{attribute 'pack_mode' := '1'} 
// ------------------------------------------------------------------------- 
//  SRCI Robot Library                                                
// ------------------------------------------------------------------------- 
//                                                                           
//  Object:      DefaultDynamics                                       
//  Author:      Thorsten Brach                                                
//  Date:        2024-06-01
//
//  Description:                                              
//   
//                                                                           
//  Copyright: 
//    (C) 2024 Thorsten Brach. All rights reserved                                                                         
//                                                                           
//  Disclaimer:                                                                           
//    This project is provided without any guarantee and can be used for   
//    private and commercial purposes. Any commercial use is at the user’s 
//    own risk and responsibility.
//
// -------------------------------------------------------------------------
TYPE DefaultDynamics :
STRUCT
  /// Timestamp
  Timestamp        : DT;
  /// Maximum velocity for the axes.
  /// Range [%]: 
  /// •  <0% : Use default velocity given by the user
  /// •   0% : Use internal minimal velocity
  /// • 100% : Use the entire reference velocity, given by the user
  VelocityRate     : REAL;
  /// Maximum acceleration.
  /// Range [%]:
  /// •  <0% : Use default acceleration given by the user
  /// •   0% : Use internal minimal acceleration
  /// • 100% : Use the entire reference acceleration, given by the user
  AccelerationRate : REAL;
  /// Maximum deceleration.
  /// Range [%] : 
  /// •  <0% : Use default deceleration given by the user
  /// •   0% : Use internal minimal deceleration
  /// • 100% : Use the entire reference deceleration, given by the user
  DecelerationRate : REAL;
  /// Maximum jerk
  /// Range [%] : 
  /// •  <0% : Use default jerk given by the user
  /// •   0% : Use internal minimal jerk
  /// • 100% : Use the entire reference jerk, given by the user (Trapezoidal if possible) 
  JerkRate         : REAL;  
END_STRUCT
END_TYPE

{attribute 'pack_mode' := '1'}
// ------------------------------------------------------------------------- 
//  SRCI Robot Library                                                
// ------------------------------------------------------------------------- 
//                                                                           
//  Object:      ReferenceDynamics                                       
//  Author:      Thorsten Brach                                                
//  Date:        2024-06-01
//
//  Description:                                              
//   
//                                                                           
//  Copyright: 
//    (C) 2024 Thorsten Brach. All rights reserved                                                                         
//                                                                           
//  Disclaimer:                                                                           
//    This project is provided without any guarantee and can be used for   
//    private and commercial purposes. Any commercial use is at the user’s 
//    own risk and responsibility.
//
// ------------------------------------------------------------------------- 
TYPE ReferenceDynamics :
STRUCT
  /// Timestamp
  Timestamp             : DT;
  /// Path velocity [mm/s](tangent) at 100%
  /// • <0: (default) - Do not change values
  /// • ≥0: Change values according to input value
  VelocityReference     : REAL;
  /// Path acceleration [mm/s2] at 100%
  /// • <0: (default) - Do not change values
  /// • ≥0: Change values according to input value
  AccelerationReference : REAL;
  /// Path deceleration [mm/s2] at 100%
  /// • <0: (default) - Do not change values
  /// • ≥0: Change values according to input value
  DecelerationReference : REAL;
  /// Jerk [mm/s3] at 100%
  /// • <0: (default) - Do not change values
  /// • ≥0: Change values according to input value
  JerkRate              : REAL;  
END_STRUCT
END_TYPE

{attribute 'pack_mode' := '1'} 
// ------------------------------------------------------------------------- 
//  SRCI Robot Library                                                
// ------------------------------------------------------------------------- 
//                                                                           
//  Object:      RobotJointCurrent                                       
//  Author:      Thorsten Brach                                                
//  Date:        2024-06-01
//
//  Description:                                              
//   
//                                                                           
//  Copyright: 
//    (C) 2024 Thorsten Brach. All rights reserved                                                                         
//                                                                           
//  Disclaimer:                                                                           
//    This project is provided without any guarantee and can be used for   
//    private and commercial purposes. Any commercial use is at the user’s 
//    own risk and responsibility.
//
// -------------------------------------------------------------------------
TYPE RobotJointCurrent :
STRUCT
  /// Current of first joint of the robot
  J1 : REAL;
  /// Current of second joint of the robot
  J2 : REAL;
  /// Current of third joint of the robot
  J3 : REAL;
  /// Current of fourth joint of the robot
  J4 : REAL;
  /// Current of fifth joint of the robot
  J5 : REAL;
  /// Current of sixth joint of the robot
  J6 : REAL;
  /// Current of first external joint of the robot
  E1 : REAL;
  /// Current of second external axis
  E2: REAL;
  /// Current of third external axis
  E3: REAL;
  /// Current of fourth external axis
  E4: REAL;
  /// Current of fifth external axis
  E5: REAL;
  /// Current of sixth external axis
  E6: REAL;  
END_STRUCT
END_TYPE

{attribute 'pack_mode' := '1'} 
// ------------------------------------------------------------------------- 
//  SRCI Robot Library                                                
// ------------------------------------------------------------------------- 
//                                                                           
//  Object:      RobotJointCurrentExt                                       
//  Author:      Thorsten Brach                                                
//  Date:        2024-06-01
//
//  Description:                                              
//   
//                                                                           
//  Copyright: 
//    (C) 2024 Thorsten Brach. All rights reserved                                                                         
//                                                                           
//  Disclaimer:                                                                           
//    This project is provided without any guarantee and can be used for   
//    private and commercial purposes. Any commercial use is at the user’s 
//    own risk and responsibility.
//
// -------------------------------------------------------------------------
TYPE RobotJointCurrentExt :
STRUCT
  /// Current of first external joint of the robot
  E1 : REAL;
  /// Current of second external axis
  E2: REAL;
  /// Current of third external axis
  E3: REAL;
  /// Current of fourth external axis
  E4: REAL;
  /// Current of fifth external axis
  E5: REAL;
  /// Current of sixth external axis
  E6: REAL;  
END_STRUCT
END_TYPE

{attribute 'pack_mode' := '1'} 
// ------------------------------------------------------------------------- 
//  SRCI Robot Library                                                
// ------------------------------------------------------------------------- 
//                                                                           
//  Object:      RobotJointCurrentShort                                       
//  Author:      Thorsten Brach                                                
//  Date:        2024-06-01
//
//  Description:                                              
//   
//                                                                           
//  Copyright: 
//    (C) 2024 Thorsten Brach. All rights reserved                                                                         
//                                                                           
//  Disclaimer:                                                                           
//    This project is provided without any guarantee and can be used for   
//    private and commercial purposes. Any commercial use is at the user’s 
//    own risk and responsibility.
//
// -------------------------------------------------------------------------
TYPE RobotJointCurrentShort :
STRUCT
  /// Current of first joint of the robot
  J1 : REAL;
  /// Current of second joint of the robot
  J2 : REAL;
  /// Current of third joint of the robot
  J3 : REAL;
  /// Current of fourth joint of the robot
  J4 : REAL;
  /// Current of fifth joint of the robot
  J5 : REAL;
  /// Current of sixth joint of the robot
  J6 : REAL;
END_STRUCT
END_TYPE

{attribute 'pack_mode' := '1'} 
// ------------------------------------------------------------------------- 
//  SRCI Robot Library                                                
// ------------------------------------------------------------------------- 
//                                                                           
//  Object:      RobotJointPosition                                       
//  Author:      Thorsten Brach                                                
//  Date:        2024-06-01
//
//  Description:                                              
//   
//                                                                           
//  Copyright: 
//    (C) 2024 Thorsten Brach. All rights reserved                                                                         
//                                                                           
//  Disclaimer:                                                                           
//    This project is provided without any guarantee and can be used for   
//    private and commercial purposes. Any commercial use is at the user’s 
//    own risk and responsibility.
//
// -------------------------------------------------------------------------
TYPE RobotJointPosition :
STRUCT
  /// Position [°] of first joint of the robot
  J1 : REAL;
  /// Position [°] of second joint of the robot
  J2 : REAL;
  /// Position [°] of third joint of the robot
  J3 : REAL;
  /// Position [°] of fourth joint of the robot
  J4 : REAL;
  /// Position [°] of fifth joint of the robot
  J5 : REAL;
  /// Position [°] of sixth joint of the robot
  J6 : REAL;
  /// Position [°] of first external axis 
  E1 : REAL;  
  /// Position [°] of second external axis
  E2 : REAL;
  /// Position [°] of third external axis
  E3 : REAL;
  /// Position [°] of fourth external axis
  E4 : REAL;
  /// Position [°] of fifth external axis
  E5 : REAL;
  /// Position [°] of sixth external axis
  E6 : REAL;  
END_STRUCT
END_TYPE

{attribute 'pack_mode' := '1'} 
// ------------------------------------------------------------------------- 
//  SRCI Robot Library                                                
// ------------------------------------------------------------------------- 
//                                                                           
//  Object:      RobotJointPositionExt                                       
//  Author:      Thorsten Brach                                                
//  Date:        2024-06-01
//
//  Description:                                              
//   
//                                                                           
//  Copyright: 
//    (C) 2024 Thorsten Brach. All rights reserved                                                                         
//                                                                           
//  Disclaimer:                                                                           
//    This project is provided without any guarantee and can be used for   
//    private and commercial purposes. Any commercial use is at the user’s 
//    own risk and responsibility.
//
// -------------------------------------------------------------------------
TYPE RobotJointPositionExt :
STRUCT
  /// Position of second external axis
  E2: REAL;
  /// Position of third external axis
  E3: REAL;
  /// Position of fourth external axis
  E4: REAL;
  /// Position of fifth external axis
  E5: REAL;
  /// Position of sixth external axis
  E6: REAL;  
END_STRUCT
END_TYPE

{attribute 'pack_mode' := '1'} 
// ------------------------------------------------------------------------- 
//  SRCI Robot Library                                                
// ------------------------------------------------------------------------- 
//                                                                           
//  Object:      RobotJointPositionShort                                       
//  Author:      Thorsten Brach                                                
//  Date:        2024-06-01
//
//  Description:                                              
//   
//                                                                           
//  Copyright: 
//    (C) 2024 Thorsten Brach. All rights reserved                                                                         
//                                                                           
//  Disclaimer:                                                                           
//    This project is provided without any guarantee and can be used for   
//    private and commercial purposes. Any commercial use is at the user’s 
//    own risk and responsibility.
//
// -------------------------------------------------------------------------
TYPE RobotJointPositionShort :
STRUCT
  /// Position of first joint of the robot
  J1 : REAL;
  /// Position of second joint of the robot
  J2 : REAL;
  /// Position of third joint of the robot
  J3 : REAL;
  /// Position of fourth joint of the robot
  J4 : REAL;
  /// Position of fifth joint of the robot
  J5 : REAL;
  /// Position of sixth joint of the robot
  J6 : REAL;
  /// Position of first external axis 
  E1 : REAL;  
END_STRUCT
END_TYPE

{attribute 'pack_mode' := '1'} 
// ------------------------------------------------------------------------- 
//  SRCI Robot Library                                                
// ------------------------------------------------------------------------- 
//                                                                           
//  Object:      AlarmMessage                                       
//  Author:      Thorsten Brach                                                
//  Date:        2024-06-01
//
//  Description:                                              
//   
//                                                                           
//  Copyright: 
//    (C) 2024 Thorsten Brach. All rights reserved                                                                         
//                                                                           
//  Disclaimer:                                                                           
//    This project is provided without any guarantee and can be used for   
//    private and commercial purposes. Any commercial use is at the user’s 
//    own risk and responsibility.
//
// -------------------------------------------------------------------------
TYPE AlarmMessage :
STRUCT
  /// Timestamp
  Timestamp   : DT;
  /// Type of message according to Table 5-46:
  MessageType : MessageType;
  /// Severity of message according to Table 5-47: Debug, Info, Warning, Error, Fatal error
  Severity    : Severity;
  /// Code of messages
  MessageCode : DWORD;
  /// Static text of message
  MessageText : STRING(150);  
END_STRUCT
END_TYPE

{attribute 'pack_mode' := '1'} 
// ------------------------------------------------------------------------- 
//  SRCI Robot Library                                                
// ------------------------------------------------------------------------- 
//                                                                           
//  Object:      ArmConfigParameter                                       
//  Author:      Thorsten Brach                                                
//  Date:        2024-06-01
//
//  Description:                                              
//   
//                                                                           
//  Copyright: 
//    (C) 2024 Thorsten Brach. All rights reserved                                                                         
//                                                                           
//  Disclaimer:                                                                           
//    This project is provided without any guarantee and can be used for   
//    private and commercial purposes. Any commercial use is at the user’s 
//    own risk and responsibility.
//
// -------------------------------------------------------------------------
TYPE ArmConfigParameter :
STRUCT
  /// Configuration of shoulder
  Shoulder : ArmConfigShoulder;
  /// Configuration of elbow
  Elbow    : ArmConfigElbow;
  /// Configuration of wrist
  Wrist    : ArmConfigWrist;
END_STRUCT
END_TYPE

{attribute 'pack_mode' := '1'} 
// ------------------------------------------------------------------------- 
//  SRCI Robot Library                                                
// ------------------------------------------------------------------------- 
//                                                                           
//  Object:      AuxOffset                                       
//  Author:      Thorsten Brach                                                
//  Date:        2024-06-01
//
//  Description:                                              
//   
//                                                                           
//  Copyright: 
//    (C) 2024 Thorsten Brach. All rights reserved                                                                         
//                                                                           
//  Disclaimer:                                                                           
//    This project is provided without any guarantee and can be used for   
//    private and commercial purposes. Any commercial use is at the user’s 
//    own risk and responsibility.
//
// -------------------------------------------------------------------------
TYPE AuxOffset :
STRUCT
  /// Offset in X-Direction
  X : REAL;
  /// Offset in Y-direction
  Y : REAL;
  /// Offset in Z-direction
  Z : REAL;
END_STRUCT
END_TYPE

{attribute 'pack_mode' := '1'} 
// ------------------------------------------------------------------------- 
//  SRCI Robot Library                                                
// ------------------------------------------------------------------------- 
//                                                                           
//  Object:      CoordinateSystem                                       
//  Author:      Thorsten Brach                                                
//  Date:        2024-06-01
//
//  Description:                                              
//   
//                                                                           
//  Copyright: 
//    (C) 2024 Thorsten Brach. All rights reserved                                                                         
//                                                                           
//  Disclaimer:                                                                           
//    This project is provided without any guarantee and can be used for   
//    private and commercial purposes. Any commercial use is at the user’s 
//    own risk and responsibility.
//
// -------------------------------------------------------------------------
TYPE CoordinateSystem :
STRUCT
  /// Tool index
  /// • 0: Flange
  /// • 1..254: Tool frames
  ToolNo  : USINT;
  /// Frame index
  /// • 0: WCS
  /// • 1..254: User frames
  FrameNo : USINT;
END_STRUCT
END_TYPE

{attribute 'pack_mode' := '1'} 
// ------------------------------------------------------------------------- 
//  SRCI Robot Library                                                
// ------------------------------------------------------------------------- 
//                                                                           
//  Object:      DataInSync                                       
//  Author:      Thorsten Brach                                                
//  Date:        2024-06-01
//
//  Description:                                              
//   
//                                                                           
//  Copyright: 
//    (C) 2024 Thorsten Brach. All rights reserved                                                                         
//                                                                           
//  Disclaimer:                                                                           
//    This project is provided without any guarantee and can be used for   
//    private and commercial purposes. Any commercial use is at the user’s 
//    own risk and responsibility.
//
// -------------------------------------------------------------------------
TYPE DataInSync :
STRUCT
  /// TRUE, if no tool has been modified
  ToolsInSync             : BOOL;
  /// TRUE, if no frame has been modified
  FramesInSync            : BOOL;
  /// TRUE, if no load has been modified
  LoadsInSync             : BOOL;
  /// TRUE, if no work area has been modified
  WorkAreasInSync         : BOOL;
  /// TRUE, if no software limit has been modified
  SoftwareLimitsInSync    : BOOL;
  /// TRUE, if no default dynamic parameter has been modified
  DefaultDynamicsInSync   : BOOL;
  /// TRUE, if no reference dynamic parameter has been modified
  ReferenceDynamicsInSync : BOOL;  
END_STRUCT
END_TYPE

{attribute 'pack_mode' := '1'} 
// ------------------------------------------------------------------------- 
//  SRCI Robot Library                                                
// ------------------------------------------------------------------------- 
//                                                                           
//  Object:      DHParameter                                       
//  Author:      Thorsten Brach                                                
//  Date:        2024-06-01
//
//  Description:                                              
//   
//                                                                           
//  Copyright: 
//    (C) 2024 Thorsten Brach. All rights reserved                                                                         
//                                                                           
//  Disclaimer:                                                                           
//    This project is provided without any guarantee and can be used for   
//    private and commercial purposes. Any commercial use is at the user’s 
//    own risk and responsibility.
//
// -------------------------------------------------------------------------
TYPE DHParameter :
STRUCT
   /// DH parameter α for each joint - 0 If not supported
   Alpha                  : ARRAY [0..6] OF REAL;
   /// DH parameters A for each joint - 0 If not supported
   A                      : ARRAY [0..6] OF REAL;
   /// DH parameters D for each joint - 0 If not supported
   D                      : ARRAY [0..6] OF REAL;
   /// DH parameters Theta for each joint - 0 If not supported
   Theta                  : ARRAY [0..6] OF REAL;
   /// Positive joint direction of each joint. TRUE when positive joint direction points to the right.
   /// See also Figure 6-16.
   PositiveJointDirection : ARRAY [0..6] OF BOOL;
   /// Offset of zero position of joint to zero position suggested by Figure 6-17.
   JointZeroPosition      : ARRAY [0..6] OF REAL;
END_STRUCT
END_TYPE

{attribute 'pack_mode' := '1'} 
// ------------------------------------------------------------------------- 
//  SRCI Robot Library                                                
// ------------------------------------------------------------------------- 
//                                                                           
//  Object:      ExternalAxesFlags                                       
//  Author:      Thorsten Brach                                                
//  Date:        2024-06-01
//
//  Description:                                              
//   
//                                                                           
//  Copyright: 
//    (C) 2024 Thorsten Brach. All rights reserved                                                                         
//                                                                           
//  Disclaimer:                                                                           
//    This project is provided without any guarantee and can be used for   
//    private and commercial purposes. Any commercial use is at the user’s 
//    own risk and responsibility.
//
// -------------------------------------------------------------------------
TYPE ExternalAxesFlags :
STRUCT
  /// Bit 00 : Not used
  Bit00   : BOOL;
  /// Bit 01 : External axis E1 - property depends of usage 
  AxisE1  : BOOL;
  /// Bit 02 : External axis E2 - property depends of usage 
  AxisE2  : BOOL;
  /// Bit 03 : External axis E3 - property depends of usage 
  AxisE3  : BOOL;
  /// Bit 04 : External axis E4 - property depends of usage 
  AxisE4  : BOOL;
  /// Bit 05 : External axis E5 - property depends of usage 
  AxisE5  : BOOL;
  /// Bit 06 : External axis E6 - property depends of usage 
  AxisE6  : BOOL;
  /// Bit 00 : Not used
  Bit07   : BOOL;
END_STRUCT
END_TYPE

{attribute 'pack_mode' := '1'} 
// ------------------------------------------------------------------------- 
//  SRCI Robot Library                                                
// ------------------------------------------------------------------------- 
//                                                                           
//  Object:      ForceStatus                                       
//  Author:      Thorsten Brach                                                
//  Date:        2024-06-01
//
//  Description:                                              
//   
//                                                                           
//  Copyright: 
//    (C) 2024 Thorsten Brach. All rights reserved                                                                         
//                                                                           
//  Disclaimer:                                                                           
//    This project is provided without any guarantee and can be used for   
//    private and commercial purposes. Any commercial use is at the user’s 
//    own risk and responsibility.
//
// -------------------------------------------------------------------------
TYPE ForceStatus :
STRUCT
  /// TRUE, while a "ForceControl" function is enabled
  ForceControlEnabled         : BOOL;
  /// TRUE, while a "ForceLimit" function is enabled
  ForceLimitEnabled           : BOOL;
  /// TRUE, while robot is adjusting its movement to apply specified force
  ApplyingForce               : BOOL;
  /// TRUE, while maximum deviation according to input parameter "MaxDeviation" is reached
  MaxDeviationReached         : BOOL;
  /// TRUE, while currently applied force/torque is identical to specified force/torque
  SpecifiedForceTorqueReached : BOOL;
  /// TRUE, while currently detected force is identical to specified force limit
  SpecifiedForceLimitReached  : BOOL;
  /// Bit 06 Reserve
  Bit06                       : BOOL;
  /// Bit 07 Reserve
  Bit07                       : BOOL;  
END_STRUCT
END_TYPE

{attribute 'pack_mode' := '1'} 
// ------------------------------------------------------------------------- 
//  SRCI Robot Library                                                
// ------------------------------------------------------------------------- 
//                                                                           
//  Object:      FragmentAction                                       
//  Author:      Thorsten Brach                                                
//  Date:        2024-06-01
//
//  Description:                                              
//   
//                                                                           
//  Copyright: 
//    (C) 2024 Thorsten Brach. All rights reserved                                                                         
//                                                                           
//  Disclaimer:                                                                           
//    This project is provided without any guarantee and can be used for   
//    private and commercial purposes. Any commercial use is at the user’s 
//    own risk and responsibility.
//
// -------------------------------------------------------------------------
TYPE FragmentAction :
STRUCT
  /// Bit 00 : Command Message is completely received – Flag to trigger processing of the payload
  Complete : BOOL;
  /// Bit 01 :(only client->server): The first message fragment of a new CMD resets (set all ACR values of this CMD ID to 0) the ACR entry
  Reset    : BOOL;
  /// Bit 02: Clears the receiving buffer by setting all of its Bytes to 0.
  Clear    : BOOL;
  /// Bit 03
  BIT03    : BOOL;
  /// Bit 04
  BIT04    : BOOL;
  /// Bit 05
  BIT05    : BOOL;
  /// Bit 06
  BIT06    : BOOL;
  /// Bit 07
  BIT07    : BOOL;  
END_STRUCT
END_TYPE

{attribute 'pack_mode' := '1'} 
// ------------------------------------------------------------------------- 
//  SRCI Robot Library                                                
// ------------------------------------------------------------------------- 
//                                                                           
//  Object:      JogControl                                       
//  Author:      Thorsten Brach                                                
//  Date:        2024-06-01
//
//  Description:                                              
//   
//                                                                           
//  Copyright: 
//    (C) 2024 Thorsten Brach. All rights reserved                                                                         
//                                                                           
//  Disclaimer:                                                                           
//    This project is provided without any guarantee and can be used for   
//    private and commercial purposes. Any commercial use is at the user’s 
//    own risk and responsibility.
//
// -------------------------------------------------------------------------
TYPE JogControl :
STRUCT
  /// Mode Frame : Movement in positive direction X of selected frame
  /// Mode Tool  : Movement in positive direction X of selected tool
  /// Mode Axes  : Movement in positive direction joint 1
  X_J1_Pos  : BOOL;
  /// Mode Frame : Movement in negative direction X of selected frame
  /// Mode Tool  : Movement in negative direction X of selected tool
  /// Mode Axes  : Movement in negative direction joint 1
  X_J1_Neg  : BOOL;
  /// Mode Frame : Movement in positive direction Y of selected frame
  /// Mode Tool  : Movement in positive direction Y of selected tool
  /// Mode Axes  : Movement in positive direction joint 2
  Y_J2_Pos  : BOOL;
  /// Mode Frame : Movement in negative direction Y of selected frame
  /// Mode Tool  : Movement in negative direction Y of selected tool
  /// Mode Axes  : Movement in negative direction joint 2
  Y_J2_Neg  : BOOL;
  /// Mode Frame : Movement in positive direction Z of selected frame
  /// Mode Tool  : Movement in positive direction Z of selected tool
  /// Mode Axes  : Movement in positive direction joint 3
  Z_J3_Pos  : BOOL;
  /// Mode Frame : Movement in negative direction Z of selected frame
  /// Mode Tool  : Movement in negative direction Z of selected tool
  /// Mode Axes  : Movement in negative direction joint 3
  Z_J3_Neg  : BOOL;
  /// Mode Frame : Movement in positive direction Rx of selected frame
  /// Mode Tool  : Movement in positive direction Rx of selected tool
  /// Mode Axes  : Movement in positive direction joint 4
  Rx_J4_Pos : BOOL;
  /// Mode Frame : Movement in negative direction Rx of selected frame
  /// Mode Tool  : Movement in negative direction Rx of selected tool
  /// Mode Axes  : Movement in negative direction joint 4
  Rx_J4_Neg : BOOL;
  /// Mode Frame : Movement in positive direction Ry of selected frame
  /// Mode Tool  : Movement in positive direction Ry of selected tool
  /// Mode Axes  : Movement in positive direction joint 5
  Ry_J5_Pos : BOOL;
  /// Mode Frame : Movement in negative direction Ry of selected frame
  /// Mode Tool  : Movement in negative direction Ry of selected tool
  /// Mode Axes  : Movement in negative direction joint 5
  Rx_J5_Neg : BOOL;
  /// Mode Frame : Movement in positive direction Rz of selected frame
  /// Mode Tool  : Movement in positive direction Rz of selected tool
  /// Mode Axes  : Movement in positive direction joint 6
  Rz_J6_Pos : BOOL;
  /// Mode Frame : Movement in negative direction Rz of selected frame
  /// Mode Tool  : Movement in negative direction Rz of selected tool
  /// Mode Axes  : Movement in negative direction joint 6
  Rz_J6_Neg : BOOL;
  /// Mode Frame : not supported
  /// Mode Tool  : not supported
  /// Mode Axes  : Movement in positive direction first external axis
  E1_Pos    : BOOL;
  /// Mode Frame : not supported
  /// Mode Tool  : not supported
  /// Mode Axes  : Movement in negative direction first external axis
  E1_Neg    : BOOL;
  /// Mode Frame : not supported
  /// Mode Tool  : not supported
  /// Mode Axes  : Movement in positive direction second external axis
  E2_Pos    : BOOL;
  /// Mode Frame : not supported
  /// Mode Tool  : not supported
  /// Mode Axes  : Movement in negative direction second external axis
  E2_Neg    : BOOL;
  /// Mode Frame : not supported
  /// Mode Tool  : not supported
  /// Mode Axes  : Movement in positive direction third external axis
  E3_Pos    : BOOL;
  /// Mode Frame : not supported
  /// Mode Tool  : not supported
  /// Mode Axes  : Movement in negative direction third external axis
  E3_Neg    : BOOL;
  /// Mode Frame : not supported
  /// Mode Tool  : not supported
  /// Mode Axes  : Movement in positive direction fourth external axis
  E4_Pos    : BOOL;
  /// Mode Frame : not supported
  /// Mode Tool  : not supported
  /// Mode Axes  : Movement in negative direction fourth external axis
  E4_Neg    : BOOL;
  /// Mode Frame : not supported
  /// Mode Tool  : not supported
  /// Mode Axes  : Movement in positive direction fifth external axis
  E5_Pos    : BOOL;
  /// Mode Frame : not supported
  /// Mode Tool  : not supported
  /// Mode Axes  : Movement in negative direction fifth external axis
  E5_Neg    : BOOL;
  /// Mode Frame : not supported
  /// Mode Tool  : not supported
  /// Mode Axes  : Movement in positive direction sixth external axis
  E6_Pos    : BOOL;
  /// Mode Frame : not supported
  /// Mode Tool  : not supported
  /// Mode Axes  : Movement in negative direction sixts external axis
  E6_Neg    : BOOL;
  
END_STRUCT
END_TYPE

{attribute 'pack_mode' := '1'} 
// ------------------------------------------------------------------------- 
//  SRCI Robot Library                                                
// ------------------------------------------------------------------------- 
//                                                                           
//  Object:      MeasuringInputResult                                       
//  Author:      Thorsten Brach                                                
//  Date:        2024-06-01
//
//  Description:                                              
//   
//                                                                           
//  Copyright: 
//    (C) 2024 Thorsten Brach. All rights reserved                                                                         
//                                                                           
//  Disclaimer:                                                                           
//    This project is provided without any guarantee and can be used for   
//    private and commercial purposes. Any commercial use is at the user’s 
//    own risk and responsibility.
//
// -------------------------------------------------------------------------
TYPE MeasuringInputResult :
STRUCT
  /// Measured robot position value at the rising edge of the digital input in selected coordinate systems (see input parameters ToolNo and FrameNo).
  MeasuredCartesianPosition :  RobotCartesianPosition;
  /// Index of tool of returned position
  /// • 0: Flange
  /// • 1..254: Tool frames
  ToolNo                    : USINT;
  /// Index of frame of returned position
  /// • 0: WCS
  /// • 1..254: User frames
  FrameNo                   : USINT;
  /// Measured robot position value at the rising edge of the digital input in Joint position.
  MeasuredJointPosition     : RobotJointPosition;
END_STRUCT
END_TYPE

{attribute 'pack_mode' := '1'} 
// ------------------------------------------------------------------------- 
//  SRCI Robot Library                                                
// ------------------------------------------------------------------------- 
//                                                                           
//  Object:      ProcessingModeAllowed                                       
//  Author:      Thorsten Brach                                                
//  Date:        2024-06-01
//
//  Description:                                              
//   
//                                                                           
//  Copyright: 
//    (C) 2024 Thorsten Brach. All rights reserved                                                                         
//                                                                           
//  Disclaimer:                                                                           
//    This project is provided without any guarantee and can be used for   
//    private and commercial purposes. Any commercial use is at the user’s 
//    own risk and responsibility.
//
// -------------------------------------------------------------------------
TYPE ProcessingModeAllowed :
STRUCT
  /// Command is buffered in sequence buffer and executed once
  BUFFERED           : BOOL;
  /// Command is buffered in sequence buffer, aborts and empties previous commands in sequence buffer, and is executed once
  ABORTING           : BOOL;
  /// Command is buffered in parallel buffer and executed once
  PARALLEL           : BOOL;
  /// Command is buffered in parallel buffer and executed repeatedly until deliberate deactivation by user
  CONTINUOUS         : BOOL;
  /// CMD execution is stopped and/or CMD is removed from the buffer
  DEACTIVATE         : BOOL;
  /// Command is buffered in sequence buffer and executed once (Trigger based)
  TRIGGER_BUFFERED   : BOOL;
  /// Command is buffered in sequence buffer, aborts and empties previous commands in sequence buffer, and is executed once (Trigger based)
  TRIGGER_ABORTING   : BOOL;
  /// Command is buffered in parallel buffer and executed once (Trigger based)
  TRIGGER_ONCE       : BOOL;
  /// Command is buffered in parallel buffer and executed repeatedly until deliberate deactivation by user (Trigger based)
  TRIGGER_CONTINUOUS : BOOL;
  /// Command is buffered and executed multiple times when triggered. The CMD remains in the buffer until removed by the user.
  TRIGGER_MULTIPLE   : BOOL;  
END_STRUCT
END_TYPE

{attribute 'pack_mode' := '1'} 
// ------------------------------------------------------------------------- 
//  SRCI Robot Library                                                
// ------------------------------------------------------------------------- 
//                                                                           
//  Object:      RaStatusWord                                       
//  Author:      Thorsten Brach                                                
//  Date:        2024-06-01
//
//  Description:                                              
//   
//                                                                           
//  Copyright: 
//    (C) 2024 Thorsten Brach. All rights reserved                                                                         
//                                                                           
//  Disclaimer:                                                                           
//    This project is provided without any guarantee and can be used for   
//    private and commercial purposes. Any commercial use is at the user’s 
//    own risk and responsibility.
//
// -------------------------------------------------------------------------
TYPE RaStatusWord :
STRUCT
  /// Bit 00: 
  /// TRUE, when robot’s axes values change due to physical movement of axes
  IsMoving                 : BOOL;
  /// Bit 01: 
  /// TRUE, when move commands buffered by the primary sequence are currently not processed
  PrimarySequencePaused    : BOOL;
  /// Bit 02: 
  /// TRUE, when robot is moving in the primary sequence, FALSE when robot leaves its position by other means
  /// Switches back to TRUE in the following two scenarios:
  /// 1. During a change to the primary sequence the current TCP position is equal to
  ///    - position when the primary sequence was left
  ///    - target position of an interrupted move command of the primary sequence (see "ReturnToPrimary": "ReturnMode" "End position" chapter 6.3.11)
  /// 2. The primary sequence is active, and the buffer is empty while a new command is buffered by the primary sequence
  /// Independent of RA state
  InPrimaryPos             : BOOL;
  /// Bit 03:
  /// Secondary sequence is active, either by user selection or by implicit behavior
  SecondarySequenceActive  : BOOL;
  /// Bit 04:
  /// TRUE, when robot is currently blending between two move commands
  IsBlending               : BOOL;
  /// Bit 05:
  /// Shows that an error acknowledgement by the client is necessary
  ErrorPending             : BOOL;
  /// Bit 06:
  /// RC is restarting
  RestartInProgress        : BOOL;
  /// Bit 07:
  /// RA power state
  Enabled                  : BOOL;
  /// Bit 08:
  /// RA sequence states: Idle, Interrupt active, Axes controlled
  Executing                : BOOL;
  /// Bit 09:
  /// Interrupted
  Interrupted              : BOOL;
  /// Bit 10 - Bit 12:
  /// Operation Mode: T1 Local, T2 Local, Auto, Auto Ext, T1 Ext, T2 Ext
  OperationMode            : OperationMode;
  /// Bit 13:
  /// TRUE, while CollisionDetection is enabled (see chapter 6.5.35) 
  CollisionDetectedEnabled : BOOL;
  /// Bit 14:
  /// TRUE, when a collision was detected while CollisionDetection is enabled
  CollisionDetected        : BOOL;
  /// Bit 15:
  /// TRUE, when the RC request a restart of the RCinduced through the functions "WriteRobotSWLimits" or "WriteSystemVariable"
  RestartRequested         : BOOL;
  /// Bit 16:
  /// RA is currently accelerating. Support of this value is returned via exchangeConfig.
  Accelerating             : BOOL;
  /// Bit 17:
  /// RA is currently decelerating. Support of this value is returned via exchangeConfig.
  Decelerating             : BOOL;
  /// Bit 18:
  /// RA is currently not accelerating nor decelerating. Support of this value is returned via exchangeConfig.
  ConstantVelocity         : BOOL;
  /// Bit 19
  Bit19                    : BOOL;
  /// Bit 20
  Bit20                    : BOOL;
  /// Bit 21
  Bit21                    : BOOL;
  /// Bit 22
  Bit22                    : BOOL;
  /// Bit 23
  Bit23                    : BOOL;
  /// Bit 24
  Bit24                    : BOOL;
  /// Bit 25
  Bit25                    : BOOL;
  /// Bit 26
  Bit26                    : BOOL;
  /// Bit 27
  Bit27                    : BOOL;
  /// Bit 28
  Bit28                    : BOOL;
  /// Bit 29
  Bit29                    : BOOL;
  /// Bit 30
  Bit30                    : BOOL;
  /// Bit 31
  Bit31                    : BOOL;  
END_STRUCT
END_TYPE

{attribute 'pack_mode' := '1'} 
// ------------------------------------------------------------------------- 
//  SRCI Robot Library                                                
// ------------------------------------------------------------------------- 
//                                                                           
//  Object:      RCSupportedFunctions                                       
//  Author:      Thorsten Brach                                                
//  Date:        2024-06-01
//
//  Description:                                              
//   
//                                                                           
//  Copyright: 
//    (C) 2024 Thorsten Brach. All rights reserved                                                                         
//                                                                           
//  Disclaimer:                                                                           
//    This project is provided without any guarantee and can be used for   
//    private and commercial purposes. Any commercial use is at the user’s 
//    own risk and responsibility.
//
// -------------------------------------------------------------------------
TYPE RCSupportedFunctions :
STRUCT
  /// Byte 00 - Bit 0  
  Reserved                   : BOOL;
  /// Byte 00 - Bit 1 
  ReadRobotData              : BOOL;
  /// Byte 00 - Bit 2  
  EnableRobot                : BOOL;
  /// Byte 00 - Bit 3  
  GroupReset                 : BOOL;
  /// Byte 00 - Bit 4  
  ReadActualPosition         : BOOL;
  /// Byte 00 - Bit 5 
  ReadActualPositionCyclic   : BOOL;
  /// Byte 00 - Bit 6  
  ExchangeConfiguration      : BOOL;
  /// Byte 00 - Bit 7  
  SetSequence                : BOOL;
  
  /// Byte 01 - Bit 0  
  ChangeSpeedOverride        : BOOL;
  /// Byte 01 - Bit 1  
  ReadMessages               : BOOL;
  /// Byte 01 - Bit 2  
  ReadRobotReferenceDynamics : BOOL;
  /// Byte 01 - Bit 3  
  WriteFrameData             : BOOL;
  /// Byte 01 - Bit 4  
  WriteToolData              : BOOL;
  /// Byte 01 - Bit 5  
  WriteLoadData              : BOOL;
  /// Byte 01 - Bit 6  
  WriteRobotReferenceDynamics: BOOL;
  /// Byte 01 - Bit 7  
  WriteRobotDefaultDynamics  : BOOL;
  
  /// Byte 02 - Bit 0  
  ReadRobotDefaultDynamics   : BOOL;
  /// Byte 02 - Bit 1  
  ReadFrameData              : BOOL;
  /// Byte 02 - Bit 2  
  ReadToolData               : BOOL;
  /// Byte 02 - Bit 3  
  ReadLoadData               : BOOL;
  /// Byte 02 - Bit 4  
  ReadRobotSWLimits          : BOOL;
  /// Byte 02 - Bit 5  
  GroupJog                   : BOOL;
  /// Byte 02 - Bit 6  
  MoveLinearAbsolute         : BOOL;
  /// Byte 02 - Bit 7  
  MoveDirectAbsolute         : BOOL;
  
  /// Byte 03 - Bit 0  
  MoveAxesAbsolute           : BOOL;
  /// Byte 03 - Bit 1  
  GroupStop                  : BOOL;
  /// Byte 03 - Bit 2
  GroupContinue              : BOOL;
  /// Byte 03 - Bit 3
  GroupInterrupt             : BOOL;
  /// Byte 03 - Bit 4
  ReturnToPrimary            : BOOL;
  /// Byte 03 - Bit 5
  MoveLinearAbsoluteJ        : BOOL;
  /// Byte 03 - Bit 6
  MoveDirectRelative         : BOOL;
  /// Byte 03 - Bit 7
  MoveAxesRelative           : BOOL;
  
  /// Byte 04 - Bit 0
  MoveCircularAbsolute       : BOOL;
  /// Byte 04 - Bit 1
  MoveCircularRelative       : BOOL;
  /// Byte 04 - Bit 2
  MoveLinearOffset           : BOOL;
  /// Byte 04 - Bit 3
  MoveDirectOffset           : BOOL;
  /// Byte 04 - Bit 4
  WaitTime                   : BOOL;
  /// Byte 04 - Bit 5
  ReadDigitalInputs          : BOOL;
  /// Byte 04 - Bit 6
  ReadDigitalOutputs         : BOOL;
  /// Byte 04 - Bit 7
  WriteDigitalOutputs        : BOOL;
  
  /// Byte 05 - Bit 0
  ReadIntegers               : BOOL;
  /// Byte 05 - Bit 1
  ReadReals                  : BOOL;
  /// Byte 05 - Bit 2
  WriteIntegers              : BOOL;
  /// Byte 05 - Bit 3
  WriteReals                 : BOOL;
  /// Byte 05 - Bit 4
  MoveLinearCam              : BOOL;
  /// Byte 05 - Bit 5
  MoveDirectCam              : BOOL;
  /// Byte 05 - Bit 6
  MoveCircularCam            : BOOL;
  /// Byte 05 - Bit 7
  SetTriggerRegister         : BOOL;
  
  /// Byte 06 - Bit 0
  SetTriggerLimit            : BOOL;
  /// Byte 06 - Bit 1
  SetTriggerUser             : BOOL;
  /// Byte 06 - Bit 2
  SetTriggerError            : BOOL;
  /// Byte 06 - Bit 3
  ReactAtTrigger             : BOOL;
  /// Byte 06 - Bit 4
  WaitForTrigger             : BOOL;
  /// Byte 06 - Bit 5
  ReadSystemVariable         : BOOL;
  /// Byte 06 - Bit 6
  WriteSystemVariable        : BOOL;
  /// Byte 06 - Bit 7
  CalculateForwardKinematic  : BOOL;
  
  /// Byte 07 - Bit 0
  CalculateInverseKinematic  : BOOL;
  /// Byte 07 - Bit 1
  CalculateCartesianPosition : BOOL;
  /// Byte 07 - Bit 2
  CalculateTool              : BOOL;
  /// Byte 07 - Bit 3
  CalculateFrame             : BOOL;
  /// Byte 07 - Bit 4
  ActivateNextCommand        : BOOL;
  /// Byte 07 - Bit 5
  ShiftPosition              : BOOL;
  /// Byte 07 - Bit 6
  CallSubprogram             : BOOL;
  /// Byte 07 - Bit 7
  MoveLinearRelative         : BOOL;
  
  /// Byte 08 - Bit 0
  WriteCallSubprogramCyclic  : BOOL;
  /// Byte 08 - Bit 1
  ReadCallSubprogramCyclic   : BOOL;
  /// Byte 08 - Bit 2
  StopSubprogram             : BOOL;
  /// Byte 08 - Bit 3
  ReadDHParameter            : BOOL;
  /// Byte 08 - Bit 4
  RestartController          : BOOL;
  /// Byte 08 - Bit 5
  ReadActualTCPVelocity      : BOOL;
  /// Byte 08 - Bit 6
  UserLogin                  : BOOL;
  /// Byte 08 - Bit 7
  SwitchLanguage             : BOOL;
  
  /// Byte 09 - Bit 0
  WriteRobotSWLimits         : BOOL;
  /// Byte 09 - Bit 1
  SetOperationMode           : BOOL;
  /// Byte 09 - Bit 2
  ReadWorkArea               : BOOL;
  /// Byte 09 - Bit 3
  WriteWorkArea              : BOOL;
  /// Byte 09 - Bit 4
  ActivateWorkArea           : BOOL;
  /// Byte 09 - Bit 5
  MonitorWorkArea            : BOOL;
  /// Byte 09 - Bit 6
  MoveApproachLinear         : BOOL;
  /// Byte 09 - Bit 7
  MoveDepartLinear           : BOOL;
  
  /// Byte 10 - Bit 0
  MoveApproachDirect         : BOOL;
  /// Byte 10 - Bit 1
  MoveDepartDirect           : BOOL;
  /// Byte 10 - Bit 2
  SearchHardstop             : BOOL;
  /// Byte 10 - Bit 3
  SearchHardstopJ            : BOOL;
  /// Byte 10 - Bit 4
  MovePickPlaceLinear        : BOOL;
  /// Byte 10 - Bit 5
  MovePickPlaceDirect        : BOOL;
  /// Byte 10 - Bit 6
  ActivateConveyorTracking   : BOOL;
  /// Byte 10 - Bit 7
  RedefineTrackingPosition   : BOOL;

  /// Byte 11 - Bit 0
  SyncToConveyor             : BOOL;
  /// Byte 11 - Bit 1
  ConfigureConveyor          : BOOL;
  /// Byte 11 - Bit 2
  MoveSuperImposed           : BOOL;
  /// Byte 11 - Bit 3
  MoveSuperImposedDynamic    : BOOL;
  /// Byte 11 - Bit 4
  ReadAnalogInput            : BOOL;
  /// Byte 11 - Bit 5
  ReadAnalogOutput           : BOOL;
  /// Byte 11 - Bit 6
  WriteAnalogOutput          : BOOL;
  /// Byte 11 - Bit 7
  MeasuringInput             : BOOL;

  /// Byte 12 - Bit 0
  AbortMeasuringInput        : BOOL;
  /// Byte 12 - Bit 1
  SetTriggerMotion           : BOOL;
  /// Byte 12 - Bit 2
  OpenBrake                  : BOOL;
  /// Byte 12 - Bit 3
  PathAccuracyMode           : BOOL;
  /// Byte 12 - Bit 4
  AvoidSingularity           : BOOL;
  /// Byte 12 - Bit 5
  ForceControl               : BOOL;
  /// Byte 12 - Bit 6
  ForceLimit                 : BOOL;
  /// Byte 12 - Bit 7
  ReadActualForce            : BOOL;
  
  /// Byte 13 - Bit 0
  BrakeTest                  : BOOL;
  /// Byte 13 - Bit 1
  SoftSwitchTCP              : BOOL;
  /// Byte 13 - Bit 2
  CreateSpline               : BOOL;
  /// Byte 13 - Bit 3
  DeleteSpline               : BOOL;
  /// Byte 13 - Bit 4
  MoveSpline                 : BOOL;
  /// Byte 13 - Bit 5
  DynamicSpline              : BOOL;
  /// Byte 13 - Bit 6
  LoadMeasurementAutomatic   : BOOL;
  /// Byte 13 - Bit 7
  LoadMeasurementSequential  : BOOL;
  
  /// Byte 14 - Bit 0
  CollisionDetection         : BOOL;
  /// Byte 14 - Bit 1
  FreeDrive                  : BOOL;
  /// Byte 14 - Bit 2
  UnitMeasurement            : BOOL;
  /// Byte 14 - Bit 3
  Byte14Bit03                : BOOL;
  /// Byte 14 - Bit 4
  Byte14Bit04                : BOOL;
  /// Byte 14 - Bit 5
  Byte14Bit05                : BOOL;
  /// Byte 14 - Bit 6
  Byte14Bit06                : BOOL;
  /// Byte 14 - Bit 7
  Byte14Bit07                : BOOL;
  
  /// Byte 15 - Bit 0
  Byte15Bit00                : BOOL;
  /// Byte 15 - Bit 1
  Byte15Bit01                : BOOL;
  /// Byte 15 - Bit 2
  Byte15Bit02                : BOOL;
  /// Byte 15 - Bit 3
  Byte15Bit03                : BOOL;
  /// Byte 15 - Bit 4
  Byte15Bit04                : BOOL;
  /// Byte 15 - Bit 5
  Byte15Bit05                : BOOL;
  /// Byte 15 - Bit 6
  Byte15Bit06                : BOOL;
  /// Byte 15 - Bit 7
  Byte15Bit07                : BOOL;

  /// Byte 16 - Bit 0
  Byte16Bit00                : BOOL;
  /// Byte 15 - Bit 1
  Byte16Bit01                : BOOL;
  /// Byte 15 - Bit 2
  Byte16Bit02                : BOOL;
  /// Byte 15 - Bit 3
  Byte16Bit03                : BOOL;
  /// Byte 15 - Bit 4
  Byte16Bit04                : BOOL;
  /// Byte 15 - Bit 5
  Byte16Bit05                : BOOL;
  /// Byte 15 - Bit 6
  Byte16Bit06                : BOOL;
  /// Byte 15 - Bit 7
  Byte16Bit07                : BOOL;
  
  /// Byte 17 - Bit 0
  Byte17Bit00                : BOOL;
  /// Byte 17 - Bit 1
  Byte17Bit01                : BOOL;
  /// Byte 17 - Bit 2
  Byte17Bit02                : BOOL;
  /// Byte 17 - Bit 3
  Byte17Bit03                : BOOL;
  /// Byte 17 - Bit 4
  Byte17Bit04                : BOOL;
  /// Byte 17 - Bit 5
  Byte17Bit05                : BOOL;
  /// Byte 17 - Bit 6
  Byte17Bit06                : BOOL;
  /// Byte 17 - Bit 7
  Byte17Bit07                : BOOL;

  /// Byte 18 - Bit 0
  Byte18Bit00                : BOOL;
  /// Byte 18 - Bit 1
  Byte18Bit01                : BOOL;
  /// Byte 18 - Bit 2
  Byte18Bit02                : BOOL;
  /// Byte 18 - Bit 3
  Byte18Bit03                : BOOL;
  /// Byte 18 - Bit 4
  Byte18Bit04                : BOOL;
  /// Byte 18 - Bit 5
  Byte18Bit05                : BOOL;
  /// Byte 18 - Bit 6
  Byte18Bit06                : BOOL;
  /// Byte 18 - Bit 7
  Byte18Bit07                : BOOL;
END_STRUCT
END_TYPE

{attribute 'pack_mode' := '1'} 
// ------------------------------------------------------------------------- 
//  SRCI Robot Library                                                
// ------------------------------------------------------------------------- 
//                                                                           
//  Object:      RobotAxesFlags                                       
//  Author:      Thorsten Brach                                                
//  Date:        2024-06-01
//
//  Description:                                              
//   
//                                                                           
//  Copyright: 
//    (C) 2024 Thorsten Brach. All rights reserved                                                                         
//                                                                           
//  Disclaimer:                                                                           
//    This project is provided without any guarantee and can be used for   
//    private and commercial purposes. Any commercial use is at the user’s 
//    own risk and responsibility.
//
// -------------------------------------------------------------------------
TYPE RobotAxesFlags :
STRUCT
  /// Bit00 : Not used
  Bit00   : BOOL;
  /// Bit01 : Robot axis J1 - property depends of usage 
  AxisJ1  : BOOL;
  /// Bit02 : Robot axis J2 - property depends of usage 
  AxisJ2  : BOOL;
  /// Bit03 : Robot axis J3 - property depends of usage 
  AxisJ3  : BOOL;
  /// Bit04 : Robot axis J4 - property depends of usage 
  AxisJ4  : BOOL;
  /// Bit05 : Robot axis J5 - property depends of usage 
  AxisJ5  : BOOL;
  /// Bit06 : Robot axis J6 - property depends of usage 
  AxisJ6  : BOOL;
  /// Bit07 : Not used
  Bit07   : BOOL;
END_STRUCT
END_TYPE

{attribute 'pack_mode' := '1'} 
// ------------------------------------------------------------------------- 
//  SRCI Robot Library                                                
// ------------------------------------------------------------------------- 
//                                                                           
//  Object:      SWLimits                                       
//  Author:      Thorsten Brach                                                
//  Date:        2024-06-01
//
//  Description:                                              
//   
//                                                                           
//  Copyright: 
//    (C) 2024 Thorsten Brach. All rights reserved                                                                         
//                                                                           
//  Disclaimer:                                                                           
//    This project is provided without any guarantee and can be used for   
//    private and commercial purposes. Any commercial use is at the user’s 
//    own risk and responsibility.
//
// -------------------------------------------------------------------------
TYPE SWLimits :
STRUCT
  /// Timestamp
  Timestamp    : DT;
  /// Negative software limit for Joint J1 [mm/°]
  J1LowerLimit : REAL;
  /// Positive software limit for Joint J1 [mm/°]
  J1UpperLimit : REAL;
  /// Negative software limit for Joint J2 [mm/°]
  J2LowerLimit : REAL;
  /// Positive software limit for Joint J2 [mm/°]
  J2UpperLimit : REAL;
  /// Negative software limit for Joint J3 [mm/°]
  J3LowerLimit : REAL;
  /// Positive software limit for Joint J3 [mm/°]
  J3UpperLimit : REAL;
  /// Negative software limit for Joint J4 [mm/°]
  J4LowerLimit : REAL;
  /// Positive software limit for Joint J4 [mm/°]
  J4UpperLimit : REAL;
  /// Negative software limit for Joint J5 [mm/°]
  J5LowerLimit : REAL;
  /// Positive software limit for Joint J5 [mm/°]
  J5UpperLimit : REAL;
  /// Negative software limit for Joint J6 [mm/°]
  J6LowerLimit : REAL;
  /// Positive software limit for Joint J6 [mm/°]
  J6UpperLimit : REAL;
  /// Negative software limit for axis E1 [mm/°]
  E1LowerLimit : REAL;
  /// Positive software limit for axis E1 [mm/°]
  E1UpperLimit : REAL;
  /// Negative software limit for axis E2 [mm/°]
  E2LowerLimit : REAL;
  /// Positive software limit for axis E2 [mm/°]
  E2UpperLimit : REAL;
  /// Negative software limit for axis E3 [mm/°]
  E3LowerLimit : REAL;
  /// Positive software limit for axis E3 [mm/°]
  E3UpperLimit : REAL;
  /// Negative software limit for axis E4 [mm/°]
  E4LowerLimit : REAL;
  /// Positive software limit for axis E4 [mm/°]
  E4UpperLimit : REAL;
  /// Negative software limit for axis E5 [mm/°]
  E5LowerLimit : REAL;
  /// Positive software limit for axis E5 [mm/°]
  E5UpperLimit : REAL;
  /// Negative software limit for axis E6 [mm/°]
  E6LowerLimit : REAL;
  /// Positive software limit for axis E6 [mm/°]
  E6UpperLimit : REAL;  
END_STRUCT
END_TYPE

{attribute 'pack_mode' := '1'} 
// ------------------------------------------------------------------------- 
//  SRCI Robot Library                                                
// ------------------------------------------------------------------------- 
//                                                                           
//  Object:      SynchronizationModes                                       
//  Author:      Thorsten Brach                                                
//  Date:        2024-06-01
//
//  Description:                                              
//   
//                                                                           
//  Copyright: 
//    (C) 2024 Thorsten Brach. All rights reserved                                                                         
//                                                                           
//  Disclaimer:                                                                           
//    This project is provided without any guarantee and can be used for   
//    private and commercial purposes. Any commercial use is at the user’s 
//    own risk and responsibility.
//
// -------------------------------------------------------------------------
TYPE SynchronizationModes :
STRUCT
 /// synchronization direction for tool
 Tool              : SyncMode;
 /// synchronization direction for frame
 Frame             : SyncMode;
 /// synchronization direction for load
 Load              : SyncMode;
 /// synchronization direction for work areas
 WorkAreas         : SyncMode;
 /// synchronization direction for SW limits
 SWLimits          : SyncMode;
 /// synchronization direction for defaul dynamics
 DefaultDynamics   : SyncMode;
 /// synchronization direction for reference dynamics 
 ReferenceDynamics : SyncMode; 
END_STRUCT
END_TYPE

{attribute 'pack_mode' := '1'} 
// ------------------------------------------------------------------------- 
//  SRCI Robot Library                                                
// ------------------------------------------------------------------------- 
//                                                                           
//  Object:      TrackingStatus                                       
//  Author:      Thorsten Brach                                                
//  Date:        2024-06-01
//
//  Description:                                              
//   
//                                                                           
//  Copyright: 
//    (C) 2024 Thorsten Brach. All rights reserved                                                                         
//                                                                           
//  Disclaimer:                                                                           
//    This project is provided without any guarantee and can be used for   
//    private and commercial purposes. Any commercial use is at the user’s 
//    own risk and responsibility.
//
// -------------------------------------------------------------------------
TYPE TrackingStatus :
STRUCT
  /// TRUE, while a "ConveyorTracking" function is enabled
  ConveyorTrackingEnabled   : BOOL;  
  /// TRUE, while robot is waiting for condition defined by "SyncInMode" after "SyncToConveyor" has been executed
  WaitingForSynchronization : BOOL;
  /// TRUE, while robot is matching the TCP’s velocity to the conveyor’s velocity
  Synchronizing             : BOOL;
  /// TRUE, while TCP is moving synchronously to conveyor
  Synchronous               : BOOL;
  /// TRUE, while robot is terminating synchronous movement
  Desynchronizing           : BOOL;
  /// TRUE, while assigned UCS is within "SyncOutZone"
  SyncOutZoneEntered        : BOOL;
  /// TRUE, when assigned UCS leaves "SyncOutZone"
  /// Reset, when robot’s synchronous movement has been stopped
  SyncOutZoneLeft           : BOOL;
  /// Not used
  NotUsed                   : BOOL;   
END_STRUCT
END_TYPE

{attribute 'pack_mode' := '1'} 
// ------------------------------------------------------------------------- 
//  SRCI Robot Library                                                
// ------------------------------------------------------------------------- 
//                                                                           
//  Object:      TurnNumber                                       
//  Author:      Thorsten Brach                                                
//  Date:        2024-06-01
//
//  Description:                                              
//   
//                                                                           
//  Copyright: 
//    (C) 2024 Thorsten Brach. All rights reserved                                                                         
//                                                                           
//  Disclaimer:                                                                           
//    This project is provided without any guarantee and can be used for   
//    private and commercial purposes. Any commercial use is at the user’s 
//    own risk and responsibility.
//
// -------------------------------------------------------------------------
TYPE TurnNumber :
STRUCT
  /// Turn number of J1
  J1Turns : SINT;
  /// Turn number of J2
  J2Turns : SINT;
  /// Turn number of J3
  J3Turns : SINT;
  /// Turn number of J4
  J4Turns : SINT;
  /// Turn number of J5
  J5Turns : SINT;
  /// Turn number of J6
  J6Turns : SINT;
  /// Turn number of E1
  E1Turns : SINT;  
END_STRUCT
END_TYPE

{attribute 'pack_mode' := '1'} 
// ------------------------------------------------------------------------- 
//  SRCI Robot Library                                                
// ------------------------------------------------------------------------- 
//                                                                           
//  Object:      VersionStruct                                       
//  Author:      Thorsten Brach                                                
//  Date:        2024-06-01
//
//  Description:                                              
//   
//                                                                           
//  Copyright: 
//    (C) 2024 Thorsten Brach. All rights reserved                                                                         
//                                                                           
//  Disclaimer:                                                                           
//    This project is provided without any guarantee and can be used for   
//    private and commercial purposes. Any commercial use is at the user’s 
//    own risk and responsibility.
//
// -------------------------------------------------------------------------
TYPE VersionStruct :
STRUCT
  /// Major version
  MajorVersion : USINT;
  /// Minor version
  MinorVersion : USINT;
  /// Patch version  
  PatchVersion : USINT;
END_STRUCT
END_TYPE

{attribute 'pack_mode' := '1'} 
// ------------------------------------------------------------------------- 
//  SRCI Robot Library                                                
// ------------------------------------------------------------------------- 
//                                                                           
//  Object:      Telegram                                       
//  Author:      Thorsten Brach                                                
//  Date:        2024-06-01
//
//  Description:                                              
//   
//                                                                           
//  Copyright: 
//    (C) 2024 Thorsten Brach. All rights reserved                                                                         
//                                                                           
//  Disclaimer:                                                                           
//    This project is provided without any guarantee and can be used for   
//    private and commercial purposes. Any commercial use is at the user’s 
//    own risk and responsibility.
//
// -------------------------------------------------------------------------
TYPE Telegram :
STRUCT
  /// PLC to Robot
  PlcToRob : TelegramPlcToRob;
  /// Robot to PLC
  RobToPlc : TelegramRobToPlc;
END_STRUCT
END_TYPE

{attribute 'pack_mode' := '1'} 
// ------------------------------------------------------------------------- 
//  SRCI Robot Library                                                
// ------------------------------------------------------------------------- 
//                                                                           
//  Object:      RobotWorkArea                                       
//  Author:      Thorsten Brach                                                
//  Date:        2024-06-01
//
//  Description:                                              
//   
//                                                                           
//  Copyright: 
//    (C) 2024 Thorsten Brach. All rights reserved                                                                         
//                                                                           
//  Disclaimer:                                                                           
//    This project is provided without any guarantee and can be used for   
//    private and commercial purposes. Any commercial use is at the user’s 
//    own risk and responsibility.
//
// -------------------------------------------------------------------------
TYPE RobotWorkArea :
STRUCT
  /// Timestamp
  Timestamp          : DT;
  /// Defines type of work area 
  AreaType           : AreaType;
  /// Defines violation condition 
  /// • FALSE (default) : Robot must not leave defined area
  /// • TRUE            : Robot must not enter defined area
  AreaMode           : BOOL := FALSE;
  /// Defines RC’s and robot’s behavior when robot violates work area 
  ReactionMode       : WorkAreaReactionMode;
  /// Specifies whether an active work area can be edited by function WriteWorkArea
  ///  TRUE            : Modification of active work area possible
  ///  FALSE (default) : Modification of active work areas not possible 
  ActiveModification : BOOL;
  /// Relates to AreaType Box, Cylinder and Sphere. 
  DefinitionMode     : DefinitionMode;
  /// Relates to AreaType Box, Cylinder and Sphere.
  /// Index of reference frame
  /// • 0: WCS (default)
  /// • 1..254: User frames 
  FrameNo            : USINT;
  /// Relates to AreaType Box, Cylinder and Sphere. 
  /// X-value of reference point in specified frame - Default: 0
  ZeroPointX         : REAL := 0;
  /// Relates to AreaType Box, Cylinder and Sphere. 
  /// Y-value of reference point in specified frame - Default: 0
  ZeroPointY         : REAL := 0;
  /// Relates to AreaType Box, Cylinder and Sphere. 
  /// Z-value of reference point in specified frame - Default: 0
  ZeroPointZ         : REAL := 0;
  /// Limit for cartesian X    
  X                  : RobotWorkAreaLimitCartesian;
  /// Limit for cartesian Y    
  Y                  : RobotWorkAreaLimitCartesian;
  /// Limit for cartesian Z    
  Z                  : RobotWorkAreaLimitCartesian;
  /// Relates to AreaType Sphere. 
  /// Radius of cylinder or sphere - Default 0
  Radius             : REAL := 0;
  /// Limits for Joint J1  
  J1Limit            : RobotWorkAreaLimitJoint;
  /// Limits for Joint J2  
  J2Limit            : RobotWorkAreaLimitJoint;
  /// Limits for Joint J3  
  J3Limit            : RobotWorkAreaLimitJoint;
  /// Limits for Joint J4  
  J4Limit            : RobotWorkAreaLimitJoint;
  /// Limits for Joint J5  
  J5Limit            : RobotWorkAreaLimitJoint;
  /// Limits for Joint J6  
  J6Limit            : RobotWorkAreaLimitJoint;
  /// Limits for Joint E1  
  E1Limit            : RobotWorkAreaLimitJoint;
  /// Limits for Joint E2  
  E2Limit            : RobotWorkAreaLimitJoint;
  /// Limits for Joint E3  
  E3Limit            : RobotWorkAreaLimitJoint;
  /// Limits for Joint E4  
  E4Limit            : RobotWorkAreaLimitJoint;
  /// Limits for Joint E5  
  E5Limit            : RobotWorkAreaLimitJoint;
  /// Limits for Joint E6  
  E6Limit            : RobotWorkAreaLimitJoint;
END_STRUCT
END_TYPE

{attribute 'pack_mode' := '1'} 
// ------------------------------------------------------------------------- 
//  SRCI Robot Library                                                
// ------------------------------------------------------------------------- 
//                                                                           
//  Object:      RobotWorkAreaLimitCartesian                                       
//  Author:      Thorsten Brach                                                
//  Date:        2024-06-01
//
//  Description:                                              
//   
//                                                                           
//  Copyright: 
//    (C) 2024 Thorsten Brach. All rights reserved                                                                         
//                                                                           
//  Disclaimer:                                                                           
//    This project is provided without any guarantee and can be used for   
//    private and commercial purposes. Any commercial use is at the user’s 
//    own risk and responsibility.
//
// -------------------------------------------------------------------------
TYPE RobotWorkAreaLimitCartesian :
STRUCT
  /// Relates to AreaType Box, Cylinder and Sphere. 
  /// Distance in negative Direction - Default 0  
  LowerLimit : REAL := 0;
  /// Relates to AreaType Box, Cylinder and Sphere.
  /// Distance in positive Direction - Default 0  
  UpperLimit : REAL := 0;
END_STRUCT
END_TYPE

{attribute 'pack_mode' := '1'} 
// ------------------------------------------------------------------------- 
//  SRCI Robot Library                                                
// ------------------------------------------------------------------------- 
//                                                                           
//  Object:      RobotWorkAreaLimitJoint                                       
//  Author:      Thorsten Brach                                                
//  Date:        2024-06-01
//
//  Description:                                              
//   
//                                                                           
//  Copyright: 
//    (C) 2024 Thorsten Brach. All rights reserved                                                                         
//                                                                           
//  Disclaimer:                                                                           
//    This project is provided without any guarantee and can be used for   
//    private and commercial purposes. Any commercial use is at the user’s 
//    own risk and responsibility.
//
// -------------------------------------------------------------------------
TYPE RobotWorkAreaLimitJoint :
STRUCT
  /// Relates to AreaType Axes. 
  /// Negative work area limit for Joint
  /// • 0 (default) : No work area restriction of joint if lower and upper limit are set to 0  
  /// • 16#FFFF_FFFF: No lower work area restrictions for Joint
  LowerLimit : REAL := 0;
  /// Relates to AreaType Axes. 
  /// positive work area limit for Joint
  /// • 0 (default) : No work area restriction of joint if lower and upper limit of are set to 0  
  /// • 16#FFFF_FFFF: No lower work area restrictions for Joint
  UpperLimit : REAL := 0;  
END_STRUCT
END_TYPE

/// Date in the format days since 1990.01.01
TYPE IEC_DATE : UINT; 
// ------------------------------------------------------------------------- 
//  SRCI Robot Library                                                
// ------------------------------------------------------------------------- 
//                                                                           
//  Object:      IEC_DATE                                       
//  Author:      Thorsten Brach                                                
//  Date:        2024-06-01
//
//  Description:                                              
//   
//                                                                           
//  Copyright: 
//    (C) 2024 Thorsten Brach. All rights reserved                                                                         
//                                                                           
//  Disclaimer:                                                                           
//    This project is provided without any guarantee and can be used for   
//    private and commercial purposes. Any commercial use is at the user’s 
//    own risk and responsibility.
//
// -------------------------------------------------------------------------
END_TYPE

/// Time in the clients time zone in the format milliseconds since start of day
TYPE IEC_TIME : TIME_OF_DAY; 
// ------------------------------------------------------------------------- 
//  SRCI Robot Library                                                
// ------------------------------------------------------------------------- 
//                                                                           
//  Object:      IEC_TIME                                       
//  Author:      Thorsten Brach                                                
//  Date:        2024-06-01
//
//  Description:                                              
//   
//                                                                           
//  Copyright: 
//    (C) 2024 Thorsten Brach. All rights reserved                                                                         
//                                                                           
//  Disclaimer:                                                                           
//    This project is provided without any guarantee and can be used for   
//    private and commercial purposes. Any commercial use is at the user’s 
//    own risk and responsibility.
//
// -------------------------------------------------------------------------
END_TYPE

{attribute 'pack_mode' := '1'} 
// ------------------------------------------------------------------------- 
//  SRCI Robot Library                                                
// ------------------------------------------------------------------------- 
//                                                                           
//  Object:      AxesGroupAcyclic                                       
//  Author:      Thorsten Brach                                                
//  Date:        2024-06-01
//
//  Description:                                              
//   
//                                                                           
//  Copyright: 
//    (C) 2024 Thorsten Brach. All rights reserved                                                                         
//                                                                           
//  Disclaimer:                                                                           
//    This project is provided without any guarantee and can be used for   
//    private and commercial purposes. Any commercial use is at the user’s 
//    own risk and responsibility.
//
// -------------------------------------------------------------------------
TYPE AxesGroupAcyclic :
STRUCT
  // Active command register 
  ActiveCommandRegister : ActiveCommandRegisterFB;
END_STRUCT
END_TYPE

{attribute 'pack_mode' := '1'} 
// ------------------------------------------------------------------------- 
//  SRCI Robot Library                                                
// ------------------------------------------------------------------------- 
//                                                                           
//  Object:      AxesGroupAcyclicAcrEntry                                       
//  Author:      Thorsten Brach                                                
//  Date:        2024-06-01
//
//  Description:                                              
//   
//                                                                           
//  Copyright: 
//    (C) 2024 Thorsten Brach. All rights reserved                                                                         
//                                                                           
//  Disclaimer:                                                                           
//    This project is provided without any guarantee and can be used for   
//    private and commercial purposes. Any commercial use is at the user’s 
//    own risk and responsibility.
//
// -------------------------------------------------------------------------
TYPE AxesGroupAcyclicAcrEntry :
STRUCT
  /// Unique indentifier 
  UniqueID   : UDINT; 
  /// State of the command entry
  State      : ActiveCommandRegisterState;  
  /// Command data ( 1 = DataToSend 2 = DataInBuffer )
  Command    : ARRAY[1..2] OF AxesGroupAcyclicAcrEntryCmdBuffer;
  /// response data ( 1 = DataRecv 2 = DataInRecvBuffer )
  Response   : ARRAY[1..2] OF AxesGroupAcyclicAcrEntryRspBuffer;
  /// Reference to the corresponding command-FB to enable a callback mechanism
  rCommandFB : REFERENCE TO RobotLibraryBaseFB;
END_STRUCT
END_TYPE

{attribute 'pack_mode' := '1'} 
// ------------------------------------------------------------------------- 
//  SRCI Robot Library                                                
// ------------------------------------------------------------------------- 
//                                                                           
//  Object:      AxesGroupAcyclicAcrEntryCmd                                       
//  Author:      Thorsten Brach                                                
//  Date:        2024-06-01
//
//  Description:                                              
//   
//                                                                           
//  Copyright: 
//    (C) 2024 Thorsten Brach. All rights reserved                                                                         
//                                                                           
//  Disclaimer:                                                                           
//    This project is provided without any guarantee and can be used for   
//    private and commercial purposes. Any commercial use is at the user’s 
//    own risk and responsibility.
//
// -------------------------------------------------------------------------
TYPE AxesGroupAcyclicAcrEntryCmd :
STRUCT 
  /// Byte 00-03: Command header
  // Header  : AxesGroupAcyclicAcrEntryCmdHeader;
  /// Payload buffer
  Payload    : AxesGroupAcyclicAcrEntryCmdBuffer;  
  /// send buffer
  SendBuffer : AxesGroupAcyclicAcrEntryCmdBuffer;
END_STRUCT
END_TYPE

{attribute 'pack_mode' := '1'} 
// ------------------------------------------------------------------------- 
//  SRCI Robot Library                                                
// ------------------------------------------------------------------------- 
//                                                                           
//  Object:      AxesGroupAcyclicAcrEntryCmdBuffer                                       
//  Author:      Thorsten Brach                                                
//  Date:        2024-06-01
//
//  Description:                                              
//   
//                                                                           
//  Copyright: 
//    (C) 2024 Thorsten Brach. All rights reserved                                                                         
//                                                                           
//  Disclaimer:                                                                           
//    This project is provided without any guarantee and can be used for   
//    private and commercial purposes. Any commercial use is at the user’s 
//    own risk and responsibility.
//
// -------------------------------------------------------------------------
TYPE AxesGroupAcyclicAcrEntryCmdBuffer :
STRUCT
  /// Buffer state
  State             : BufferStateCmd;
  ///
  //OrderNumber       : ARRAY[0..1] OF UDINT;
  /// Payload defined by type per CMD definition. Processed by Appl. Layer Task.
  Payload           : ARRAY[0..RobotLibraryParameter.TELEGRAM_PAYLOAD_MAX] OF BYTE;
  /// Payload length
  PayloadLen        : UDINT;  
  /// Payload poiner position   
  PayLoadPtr        : DWORD;
END_STRUCT
END_TYPE

{attribute 'pack_mode' := '1'} 
// ------------------------------------------------------------------------- 
//  SRCI Robot Library                                                
// ------------------------------------------------------------------------- 
//                                                                           
//  Object:      AxesGroupAcyclicAcrEntryCmdHeader                                       
//  Author:      Thorsten Brach                                                
//  Date:        2024-06-01
//
//  Description:                                              
//   
//                                                                           
//  Copyright: 
//    (C) 2024 Thorsten Brach. All rights reserved                                                                         
//                                                                           
//  Disclaimer:                                                                           
//    This project is provided without any guarantee and can be used for   
//    private and commercial purposes. Any commercial use is at the user’s 
//    own risk and responsibility.
//
// -------------------------------------------------------------------------
TYPE AxesGroupAcyclicAcrEntryCmdHeader :
STRUCT
  /// Byte 00-01 :  CMD type as per specification
  CmdType      : CmdType;
  /// Byte 02  : ExecutionMode (Bit 0..3)
  ExecMode     : ExecutionMode;  
  /// Byte 03 : CMD priority (Bit 0..3)
  Prio         : PriorityLevel;
  /// Byte 03 : Parameter Sequence (Bit 4..7 )
  ParSeq       : BYTE;
END_STRUCT
END_TYPE

{attribute 'pack_mode' := '1'} 
// ------------------------------------------------------------------------- 
//  SRCI Robot Library                                                
// ------------------------------------------------------------------------- 
//                                                                           
//  Object:      AxesGroupAcyclicAcrEntryCmdTrigger                                       
//  Author:      Thorsten Brach                                                
//  Date:        2024-06-01
//
//  Description:                                              
//   
//                                                                           
//  Copyright: 
//    (C) 2024 Thorsten Brach. All rights reserved                                                                         
//                                                                           
//  Disclaimer:                                                                           
//    This project is provided without any guarantee and can be used for   
//    private and commercial purposes. Any commercial use is at the user’s 
//    own risk and responsibility.
//
// -------------------------------------------------------------------------
TYPE AxesGroupAcyclicAcrEntryCmdTrigger :
STRUCT
  /// Trigger related EmitterID
  EmitterID    : ARRAY[0..3] OF SINT;
  /// Trigger related ListenerID 
  ListenerID   : SINT;
  /// Reserver
  Reserve      : BYTE;
END_STRUCT
END_TYPE

{attribute 'pack_mode' := '1'} 
// ------------------------------------------------------------------------- 
//  SRCI Robot Library                                                
// ------------------------------------------------------------------------- 
//                                                                           
//  Object:      AxesGroupAcyclicAcrEntryRsp                                       
//  Author:      Thorsten Brach                                                
//  Date:        2024-06-01
//
//  Description:                                              
//   
//                                                                           
//  Copyright: 
//    (C) 2024 Thorsten Brach. All rights reserved                                                                         
//                                                                           
//  Disclaimer:                                                                           
//    This project is provided without any guarantee and can be used for   
//    private and commercial purposes. Any commercial use is at the user’s 
//    own risk and responsibility.
//
// -------------------------------------------------------------------------
TYPE AxesGroupAcyclicAcrEntryRsp :
STRUCT
  /// Byte 00-03: Header
  Header : AxesGroupAcyclicAcrEntryRspHeader;
  /// Byte 04-07: Trigger sub header
  Trigger : AxesGroupAcyclicAcrEntryRspTrigger;
  /// Byte 08-xx: RSP Payload defined by type per CMD definition. Generated by Appl. Layer Task
  Payload : ARRAY[0..RobotLibraryParameter.TELEGRAM_PAYLOAD_MAX] OF BYTE;    
END_STRUCT
END_TYPE

{attribute 'pack_mode' := '1'} 
// ------------------------------------------------------------------------- 
//  SRCI Robot Library                                                
// ------------------------------------------------------------------------- 
//                                                                           
//  Object:      AxesGroupAcyclicAcrEntryRspBuffer                                       
//  Author:      Thorsten Brach                                                
//  Date:        2024-06-01
//
//  Description:                                              
//   
//                                                                           
//  Copyright: 
//    (C) 2024 Thorsten Brach. All rights reserved                                                                         
//                                                                           
//  Disclaimer:                                                                           
//    This project is provided without any guarantee and can be used for   
//    private and commercial purposes. Any commercial use is at the user’s 
//    own risk and responsibility.
//
// -------------------------------------------------------------------------
TYPE AxesGroupAcyclicAcrEntryRspBuffer :
STRUCT
  ///
  State             : BufferStateRsp;
  ///
  //OrderNumber       : ARRAY[0..1] OF UDINT;
  /// Payload defined by type per CMD definition. Processed by Appl. Layer Task.
  Payload           : ARRAY[0..RobotLibraryParameter.TELEGRAM_PAYLOAD_MAX] OF BYTE;
  /// Payload length
  PayloadLen        : UDINT;  
  /// Payload poiner   
  PayLoadPtr        : DWORD;
END_STRUCT
END_TYPE

{attribute 'pack_mode' := '1'} 
// ------------------------------------------------------------------------- 
//  SRCI Robot Library                                                
// ------------------------------------------------------------------------- 
//                                                                           
//  Object:      AxesGroupAcyclicAcrEntryRspHeader                                       
//  Author:      Thorsten Brach                                                
//  Date:        2024-06-01
//
//  Description:                                              
//   
//                                                                           
//  Copyright: 
//    (C) 2024 Thorsten Brach. All rights reserved                                                                         
//                                                                           
//  Disclaimer:                                                                           
//    This project is provided without any guarantee and can be used for   
//    private and commercial purposes. Any commercial use is at the user’s 
//    own risk and responsibility.
//
// -------------------------------------------------------------------------
TYPE AxesGroupAcyclicAcrEntryRspHeader :
STRUCT
  /// Byte 00 : State  (Bit 0..3)
  State                : CmdMessageState; // ToDo : nicht sicher ob das richtig ist 
  /// Byte 00 : ParSeq (Bit 4..5)
  ParSeq               : BYTE;
  /// Byte 01 : Alarm Message Severity
  AlarmMessageSeverity : Severity;
  /// Byte 02 : Alarm Message Code
  AlarmMessageCode     : UINT;  
END_STRUCT
END_TYPE

{attribute 'pack_mode' := '1'} 
// ------------------------------------------------------------------------- 
//  SRCI Robot Library                                                
// ------------------------------------------------------------------------- 
//                                                                           
//  Object:      AxesGroupAcyclicAcrEntryRspTrigger                                       
//  Author:      Thorsten Brach                                                
//  Date:        2024-06-01
//
//  Description:                                              
//   
//                                                                           
//  Copyright: 
//    (C) 2024 Thorsten Brach. All rights reserved                                                                         
//                                                                           
//  Disclaimer:                                                                           
//    This project is provided without any guarantee and can be used for   
//    private and commercial purposes. Any commercial use is at the user’s 
//    own risk and responsibility.
//
// -------------------------------------------------------------------------
TYPE AxesGroupAcyclicAcrEntryRspTrigger :
STRUCT
  /// Number of Trigger based CMD invocations
  InvocationCounter       : USINT;
  /// Number of missed Triggers
  MissedInvocationCounter : USINT;
  /// FollowID of Trigger initiator
  OriginID                : WORD;
END_STRUCT
END_TYPE

{attribute 'pack_mode' := '1'} 
// ------------------------------------------------------------------------- 
//  SRCI Robot Library                                                
// ------------------------------------------------------------------------- 
//                                                                           
//  Object:      AxesGroupAcyclicExecutionOrderList                                       
//  Author:      Thorsten Brach                                                
//  Date:        2024-06-01
//
//  Description:                                              
//   
//                                                                           
//  Copyright: 
//    (C) 2024 Thorsten Brach. All rights reserved                                                                         
//                                                                           
//  Disclaimer:                                                                           
//    This project is provided without any guarantee and can be used for   
//    private and commercial purposes. Any commercial use is at the user’s 
//    own risk and responsibility.
//
// -------------------------------------------------------------------------
TYPE AxesGroupAcyclicExecutionOrderList :
STRUCT
  /// Command
  Command  : ARRAY [1..RobotLibraryParameter.ACTIVE_CMD_REGISTER_ENTRIES_MAX] OF UINT;
  /// Response
  Response : ARRAY [1..RobotLibraryParameter.ACTIVE_CMD_REGISTER_ENTRIES_MAX] OF UINT;
END_STRUCT
END_TYPE

{attribute 'pack_mode' := '1'} 
// ------------------------------------------------------------------------- 
//  SRCI Robot Library                                                
// ------------------------------------------------------------------------- 
//                                                                           
//  Object:      AxesGroupCyclicOptionalData                                       
//  Author:      Thorsten Brach                                                
//  Date:        2024-06-01
//
//  Description:                                              
//   
//                                                                           
//  Copyright: 
//    (C) 2024 Thorsten Brach. All rights reserved                                                                         
//                                                                           
//  Disclaimer:                                                                           
//    This project is provided without any guarantee and can be used for   
//    private and commercial purposes. Any commercial use is at the user’s 
//    own risk and responsibility.
//
// -------------------------------------------------------------------------
TYPE AxesGroupCyclicOptionalData :
STRUCT
  /// Optional cyclic data from PLC to Robot
  PlcToRob : AxesGroupCyclicOptionalDataPlcToRob;
  /// Optional cyclic data from Robot to PLC
  RobToPlc : AxesGroupCyclicOptionalDataRobToPlc;
END_STRUCT
END_TYPE

